# EPICS substitutions: support/ebrick/2-2-3/iocBoot/iocebrick/ebrickRMMDAC.substitutions
file ../../db/ebrDAC.db
{
pattern
{P         H       F       D       PREC    CH  MIN     MAX     PORT }

{ebrick:   rmm01:  ana01:  ao01    3       0   -10     10      RMMDAC}
{ebrick:   rmm01:  ana01:  ao02    3       1   -10     10      RMMDAC}
{ebrick:   rmm01:  ana01:  ao03    3       2   -10     10      RMMDAC}
{ebrick:   rmm01:  ana01:  ao04    3       3   -10     10      RMMDAC}

}
